PROGRAM MAIN
VAR
END_VAR

END_PROGRAM

(* stored: Version 1.1.0.1
   POU MAIN: Id {ac1e37e4-793e-4297-96ae-c58896c5bc66} *)
